FUNCTION_BLOCK WStringComparer EXTENDS Object IMPLEMENTS IComparer
VAR
	_ClassName : STRING := __POUNAME();
END_VAR

{attribute 'monitoring' := 'call'}
PROPERTY ClassName : STRING
GET
ClassName := _ClassName;
END_GET
END_PROPERTY

{attribute "object_name" := "Compare"}
METHOD Compare : COMPARISION_RESULT
VAR_INPUT
	left : PVOID;
	right : PVOID;
END_VAR
VAR
	leftPointer : POINTER TO WSTRING(255); 
	rightPointer : POINTER TO WSTRING(255); 
END_VAR
IF left = 0 AND right = 0 THEN
	Compare := COMPARISION_RESULT.EQUALS;
	RETURN;
END_IF

IF left = 0 THEN
	Compare := COMPARISION_RESULT.LEFT_LESS_RIGHT;
	RETURN;	
END_IF

IF right = 0 THEN
	Compare := COMPARISION_RESULT.LEFT_GREATER_RIGHT;
	RETURN;	
END_IF

leftPointer := left;
rightPointer := right;

IF leftPointer^ < rightPointer^ THEN
	Compare := COMPARISION_RESULT.LEFT_LESS_RIGHT;
ELSIF leftPointer^ > rightPointer^ THEN
	Compare := COMPARISION_RESULT.LEFT_GREATER_RIGHT;
ELSE
	Compare := COMPARISION_RESULT.EQUALS;	
END_IF
END_METHOD

END_FUNCTION_BLOCK

(* stored: Version 1.1.0.1
   POU WStringComparer: Id {39daa709-83c0-4275-b00a-5baf8ed9a0e2}, SpecialFunc None
   Property ClassName: Id {aaa8fa4f-15aa-42fc-b91c-184bd53ea850}
   Get Get: Id {09651e74-8174-466f-9274-bc96b7d40603}
   Method Compare: Id {0a8a8bd9-06ea-4c3f-9037-e388eb451768} *)
